// TIA Portal project "Project1" (V15.1)

(* hardware
DEVICE "S7300/ET200M station_1"  S7-300 station
   slot 0: "Rail_0"  Rail  6ES7 390-1***0-0AA0
   slot 2: "PLC_1"  CPU 312  6ES7 312-1AE13-0AB0  V2.6
      slot 0: "MPI interface_1"  X1
*)

// ===== PLC "PLC_1"  CPU 312 =====

VAR_GLOBAL   // PLC tag table "Default tag table"
   "Uklj_kon_1_out" AT %Q4.0 : Bool;
   "Uklj_kon_2_out" AT %Q4.1 : Bool;
   "Rucni rezim rada" AT %M0.0 : Bool;
   "Tag_1" AT %M0.1 : Bool;
   "Tag_2" AT %M0.2 : Bool;
   "Automatski režim rada prve pumpe" AT %M0.3 : Bool;
   "Automatski režim rada druge pumpe" AT %M0.4 : Bool;
   "Tag_3" AT %M0.5 : Bool;
   "Tag_4" AT %M1.0 : Bool;
   "Tag_5" AT %M1.1 : Bool;
   "Tag_6" AT %M0.6 : Bool;
   "Tag_7" AT %M1.2 : Bool;
   "Tag_8" AT %M1.3 : Bool;
   "Tag_9" AT %M1.4 : Bool;
   "Tag_10" AT %M2.0 : Bool;
   "Tag_11" AT %M2.1 : Bool;
   "Tag_12" AT %M2.2 : Bool;
END_VAR

DATA_BLOCK "Data_block_1"   // DB10
{ S7_Optimized_Access := 'FALSE' }
VERSION : 0.1
   VAR
      Start_1 : Bool;
      Stop_1 : Bool;
      Start_2 : Bool;
      Stop_2 : Bool;
      Auto_man : Bool;
      Br_uklj_P1 : Word;
      Br_uklj_P2 : Word;
   END_VAR
BEGIN
END_DATA_BLOCK

FUNCTION "Mode" : Void   // FC1, LAD
{ S7_Optimized_Access := 'FALSE' }
VERSION : 0.1
   VAR_TEMP   // added for the SCL form of the ladder/FBD networks
      _w1 : Bool;
      _w2 : Bool;
   END_VAR
BEGIN

REGION Network 1: Uključenje prve pumpe
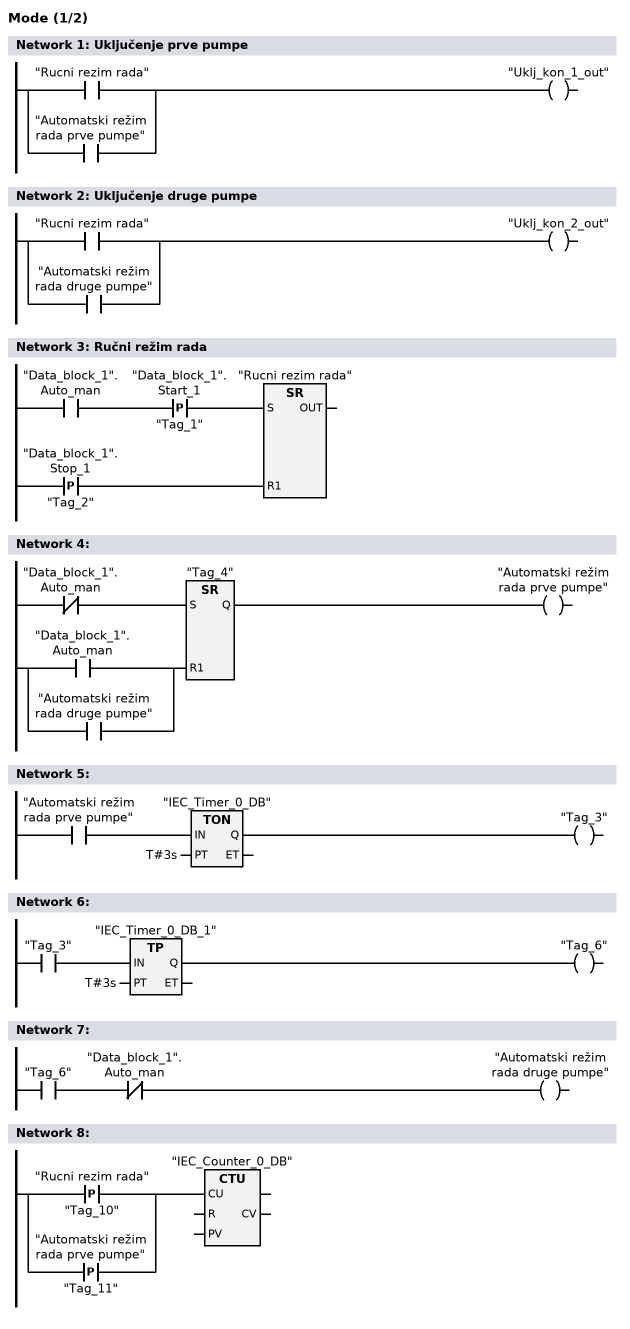
   RUNG wire#powerrail
      Contact( "Rucni rezim rada" )
      wire#w1
      Coil( "Uklj_kon_1_out" )
   END_RUNG
   RUNG wire#powerrail
      Contact( "Automatski režim rada prve pumpe" )
   END_RUNG wire#w1
   // the same network as SCL:
   "Uklj_kon_1_out" := "Rucni rezim rada" OR "Automatski režim rada prve pumpe";
END_REGION

REGION Network 2: Uključenje druge pumpe
   RUNG wire#powerrail
      Contact( "Rucni rezim rada" )
      wire#w1
      Coil( "Uklj_kon_2_out" )
   END_RUNG
   RUNG wire#powerrail
      Contact( "Automatski režim rada druge pumpe" )
   END_RUNG wire#w1
   // the same network as SCL:
   "Uklj_kon_2_out" := "Rucni rezim rada" OR "Automatski režim rada druge pumpe";
END_REGION

REGION Network 3: Ručni režim rada
   RUNG wire#powerrail
      Contact( "Data_block_1".Auto_man )
      P_Contact(operand := "Data_block_1".Start_1, bit := "Tag_1")
      S_SR(operand := "Rucni rezim rada", r1 := wire#w1)
   END_RUNG
   RUNG wire#powerrail
      P_Contact(operand := "Data_block_1".Stop_1, bit := "Tag_2")
   END_RUNG wire#w1
   // the same network as SCL:
   #_w1 := "Data_block_1".Auto_man AND "Data_block_1".Start_1 AND NOT "Tag_1";   // rising edge of "Data_block_1".Start_1
   "Tag_1" := "Data_block_1".Start_1;
   #_w2 := "Data_block_1".Stop_1 AND NOT "Tag_2";   // rising edge of "Data_block_1".Stop_1
   "Tag_2" := "Data_block_1".Stop_1;
   IF #_w1 THEN
       "Rucni rezim rada" := TRUE;   // SR flip-flop
   END_IF;
   IF #_w2 THEN "Rucni rezim rada" := FALSE; END_IF;
END_REGION

REGION Network 4
   RUNG wire#powerrail
      I_Contact( "Data_block_1".Auto_man )
      S_SR(operand := "Tag_4", r1 := wire#w1)
      Coil( "Automatski režim rada prve pumpe" )
   END_RUNG
   RUNG wire#powerrail
      Contact( "Data_block_1".Auto_man )
   END_RUNG wire#w1
   RUNG wire#powerrail
      Contact( "Automatski režim rada druge pumpe" )
   END_RUNG wire#w1
   // the same network as SCL:
   IF NOT "Data_block_1".Auto_man THEN
       "Tag_4" := TRUE;   // SR flip-flop
   END_IF;
   IF "Data_block_1".Auto_man OR "Automatski režim rada druge pumpe" THEN "Tag_4" := FALSE; END_IF;
   "Automatski režim rada prve pumpe" := "Tag_4";
END_REGION

REGION Network 5
   "IEC_Timer_0_DB".TON(IN := "Automatski režim rada prve pumpe", PT := T#3s);
   "Tag_3" := "IEC_Timer_0_DB".Q;
END_REGION

REGION Network 6
   "IEC_Timer_0_DB_1".TP(IN := "Tag_3", PT := T#3s);
   "Tag_6" := "IEC_Timer_0_DB_1".Q;
END_REGION

REGION Network 7
   RUNG wire#powerrail
      Contact( "Tag_6" )
      I_Contact( "Data_block_1".Auto_man )
      Coil( "Automatski režim rada druge pumpe" )
   END_RUNG
   // the same network as SCL:
   "Automatski režim rada druge pumpe" := "Tag_6" AND NOT "Data_block_1".Auto_man;
END_REGION

REGION Network 8
   #_w1 := "Rucni rezim rada" AND NOT "Tag_10";   // rising edge of "Rucni rezim rada"
   "Tag_10" := "Rucni rezim rada";
   #_w2 := "Automatski režim rada prve pumpe" AND NOT "Tag_11";   // rising edge of "Automatski režim rada prve pumpe"
   "Tag_11" := "Automatski režim rada prve pumpe";
   "IEC_Counter_0_DB".CTU(CU := #_w1 OR #_w2);
END_REGION

REGION Network 9
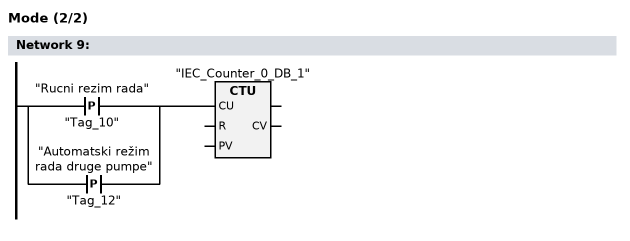
   #_w1 := "Rucni rezim rada" AND NOT "Tag_10";   // rising edge of "Rucni rezim rada"
   "Tag_10" := "Rucni rezim rada";
   #_w2 := "Automatski režim rada druge pumpe" AND NOT "Tag_12";   // rising edge of "Automatski režim rada druge pumpe"
   "Tag_12" := "Automatski režim rada druge pumpe";
   "IEC_Counter_0_DB_1".CTU(CU := #_w1 OR #_w2);
END_REGION
END_FUNCTION

ORGANIZATION_BLOCK "Main"   // OB1, LAD
TITLE = "Main Program Sweep (Cycle)"
{ S7_Optimized_Access := 'FALSE' }
VERSION : 0.1
   VAR_TEMP
      OB1_EV_CLASS : Byte;   // Bits 0-3 = 1 (Coming event), Bits 4-7 = 1 (Event class 1)
      OB1_SCAN_1 : Byte;   // 1 (Cold restart scan 1 of OB 1), 3 (Scan 2-n of OB 1)
      OB1_PRIORITY : Byte;   // Priority of OB Execution
      OB1_OB_NUMBR : Byte;   // 1 (Organization block 1, OB1)
      OB1_RESERVED_1 : Byte;   // Reserved for system
      OB1_RESERVED_2 : Byte;   // Reserved for system
      OB1_PREV_CYCLE : Int;   // Cycle time of previous OB1 scan (milliseconds)
      OB1_MIN_CYCLE : Int;   // Minimum cycle time of OB1 (milliseconds)
      OB1_MAX_CYCLE : Int;   // Maximum cycle time of OB1 (milliseconds)
      OB1_DATE_TIME : Date_And_Time;   // Date and time OB1 started
   END_VAR
BEGIN

REGION Network 1
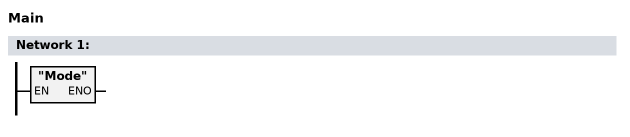
   RUNG wire#powerrail
      "Mode"()
   END_RUNG
   // the same network as SCL:
   "Mode"();
END_REGION
END_ORGANIZATION_BLOCK